Fanuc TP program (LS listing): _BOOT.LS

/PROG  _BOOT
/ATTR
OWNER		= MNEDITOR;
COMMENT		= "";
PROG_SIZE	= 199;
CREATE		= DATE 16-12-02  TIME 22:01:34;
MODIFIED	= DATE 16-12-02  TIME 22:27:24;
FILE_NAME	= ;
VERSION		= 0;
LINE_COUNT	= 2;
MEMORY_SIZE	= 571;
PROTECT		= READ_WRITE;
TCD:  STACK_SIZE	= 0,
      TASK_PRIORITY	= 50,
      TIME_SLICE	= 0,
      BUSY_LAMP_OFF	= 1,
      ABORT_REQUEST	= 7,
      PAUSE_REQUEST	= 7;
DEFAULT_GROUP	= *,*,*,*,*;
CONTROL_CODE	= 00000000 00000000;
/APPL
/APPL

AUTO_SINGULARITY_HEADER;
  ENABLE_SINGULARITY_AVOIDANCE   : TRUE;
/MN
   1:  WAIT   5.00(sec) ;
   2:  RUN _BG_SCANNERS ;
/POS
/END
